FUNCTION_BLOCK ATest
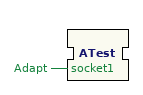
  SOCKETS
    socket1 : Adapt;
  END_SOCKETS
  EC_STATES
    START;
  END_STATES
  ALGORITHM A1 IN ST:

  END_ALGORITHM
END_FUNCTION_BLOCK
